TYPE ST_CM_Settings :
(**************************************************************************************
 * 	Application		:	BoxControl Framework
 *	Revision		:	$Revision: 404529 $
 *	Revision date	:	$Date: 2018-04-23 08:21:38 +0200 (Mo., 23 Apr 2018) $
 *	Last changed by	:	$Author: b7bolm $
 *	URL				:	$URL: http://almscdc.swisslog.com/repo/SWPD/Development/BoxControlFramework/20_Release/trunk/01_Software/BCF/BCF/JumpStart/20_Product/10_App/10_Base/10_Lib/01_DUTs/ST_CM_Settings.TcDUT $
 *
 *	Purpose			:	Condition Monitor Variable Settings Set via Telegram					
 *
 *
 * ------------------------------------------------------------------------------------
 *	Copyright Swisslog [IP AG], Switzerland. All rights reserved.
 * 
 * ------------------------------------------------------------------------------------
 *	
 * 	Revision History: 
 *
 * 	VERSION			DATE			INITIALS			DESCRIPTION
 *	0.1				01.01.2001		swl					Example
 *
 **************************************************************************************)	
STRUCT
	mVariableName		: STRING(System.CM_VARIABLENAME_STRINGLENGTH); //Variable Name 
	MaxReportTime		: TIME; // Maximum RpertTime hh:mm:ss	Default:’00:00:00’ = off
	SampleTime			: TIME; // Sample Report Time hh:mm:ss.SSS
	Threshold			: INT;  // Threshold – Minimum value change to capture a new value
	Option				: BOOL; //  Self-reset = FALSE , Reset forbidden:= True
	Enable				: BOOL; // Enable Logging 
	ErrorCode			: INT;  // Error Code 
END_STRUCT
END_TYPE

(* stored: Version 1.1.0.1, ProductVersion 3.1.4022.12
   DUT ST_CM_Settings: Id {f932e9bb-4b47-473f-b593-92f804808aa4} *)
